Fanuc KAREL source: ka00121.KL

-- PROVISIONAL review KL for V940-1; original PC SHA256 3f81130c0e4f423d73ed3e9f16a8001f38fff41aca7accf365f41d9f039c809b
-- Incomplete behavior may be omitted. Consult companion uncertainty JSON. Do not deploy.
PROGRAM KA00121
%NOLOCKGROUP
VAR
  DST : INTEGER
-- UNRESOLVED_DECL SRC type=002018
BEGIN
  -- V9_ZERO_TABLE_METADATA_HINT layout=0001; no indexed target words; source/name/runtime held
  -- UNRESOLVED_PC offsets 5-19; opcodes 2E,22,9D,33,B2
  -- UNRESOLVED_PC offsets 24-39; opcodes 22,9D,33,B1,23
  -- UNRESOLVED_PC offsets 44-48; opcodes 7F
END KA00121
